(* PLC project Unnamed, Unknown Unnamed 1 *)
(* stored: creationDateTime 2022-08-16T15:49:17, modificationDateTime 2024-04-10T21:29:34 *)

PROGRAM ArduinoPrint
  VAR
    blink_led AT %QX0.3 : BOOL;
  END_VAR
  VAR
    TON0 : TON;
    TOF0 : TOF;
  END_VAR
  VAR_EXTERNAL
    SerialMSG : STRING;
    PrintMSG : BOOL;
  END_VAR
  VAR  (* added by the conversion: wires and edge detectors of the diagram *)
    R_TRIG1 : R_TRIG;
  END_VAR

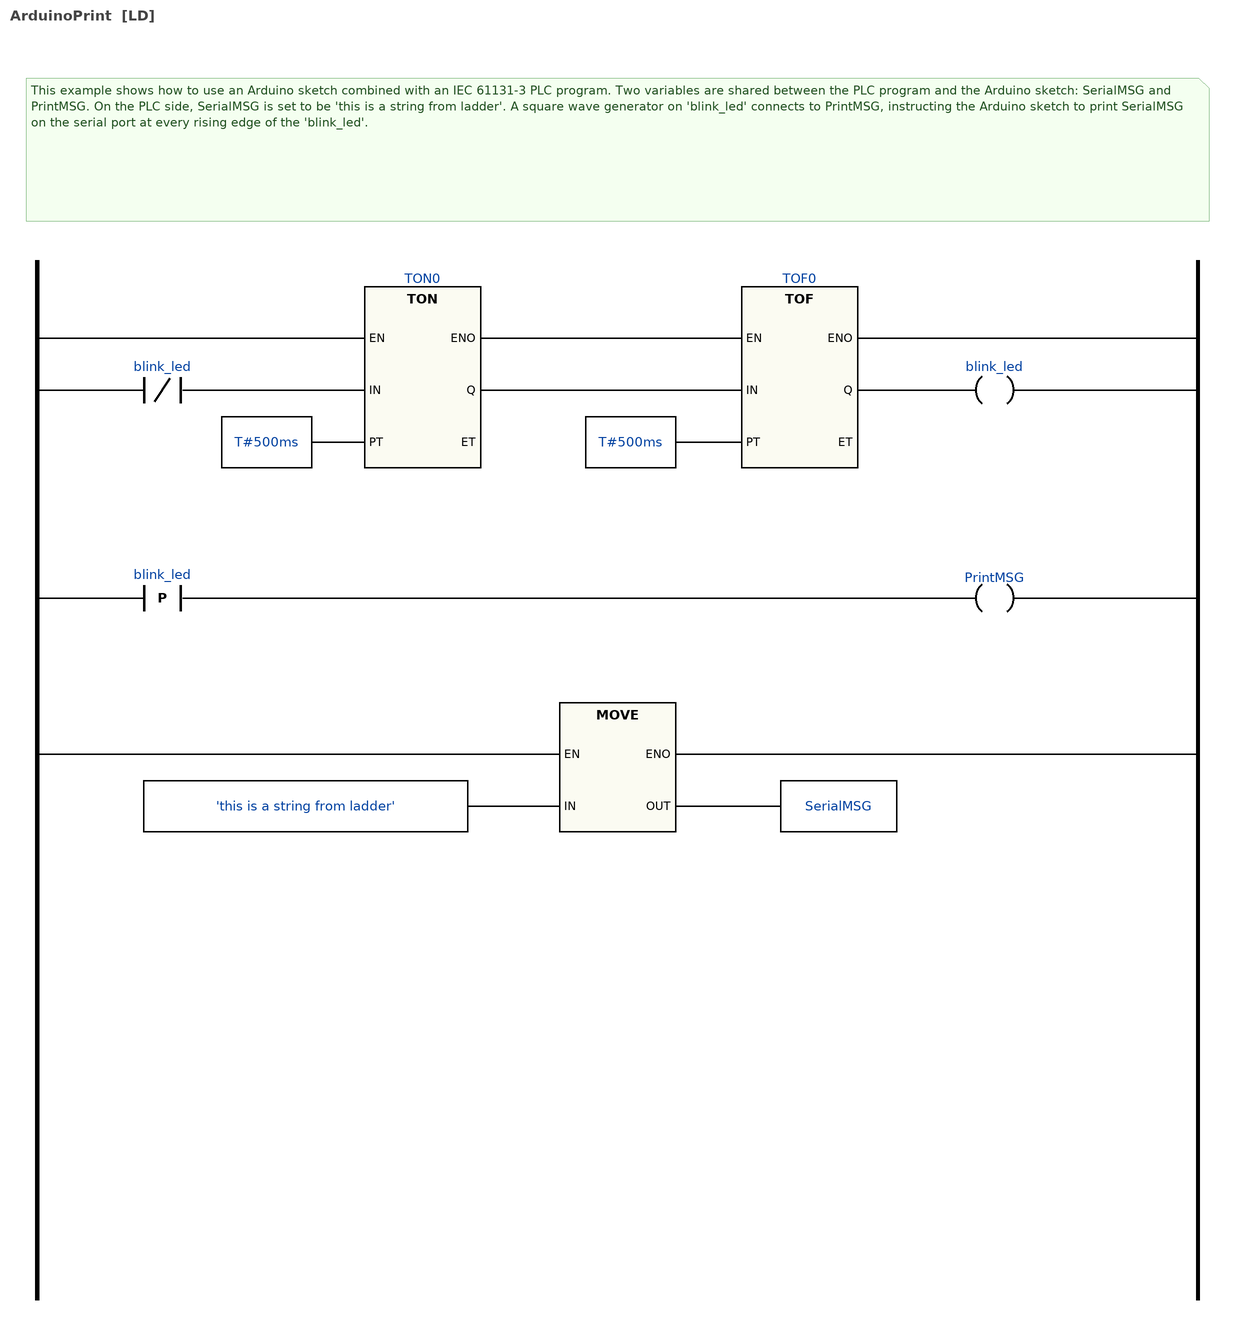
(* LD diagram, written out as Structured Text *)
(* This example shows how to use an Arduino sketch combined with an IEC 61131-3 PLC program. Two variables are shared between the PLC program and the Arduino sketch: SerialMSG and PrintMSG. On the PLC side, SerialMSG is set to be 'this is a string from ladder'. A square wave generator on 'blink_led' connects to PrintMSG, instructing the Arduino sketch to print SerialMSG on the serial port at every rising edge of the 'blink_led'. *)
TON0(IN := NOT blink_led, PT := T#500ms);
TOF0(EN := TON0.ENO, IN := TON0.Q, PT := T#500ms);
blink_led := TOF0.Q;
R_TRIG1(CLK := blink_led);
PrintMSG := R_TRIG1.Q;
SerialMSG := 'this is a string from ladder';
END_PROGRAM

CONFIGURATION Config0
  RESOURCE Res0 ON PLC
    TASK task0(INTERVAL := T#20ms, PRIORITY := 0);
    PROGRAM instance0 WITH task0 : ArduinoPrint;
  END_RESOURCE
END_CONFIGURATION
